// TIA Portal V20 export
TYPE "typeUnitCommunicationControlNode"
// stored: Namespace Unit1.Em2
   STRUCT
      BA030 : "Unit1.Em2.typeUnitCommunicationControlNodeBA030";
      BA040 : "Unit1.Em2.typeUnitCommunicationControlNodeBA040";
   END_STRUCT;
END_TYPE
